FUNCTION_BLOCK FB_Idle IMPLEMENTS I_State
VAR_INPUT
	(* Pointer to the ATM Machine*)
	pATM_Machine	: POINTER TO FB_ATM_Machine;
END_VAR
VAR_OUTPUT
END_VAR
VAR
END_VAR

METHOD Cancel : BOOL
END_METHOD

METHOD Card_Ejected : BOOL
END_METHOD

METHOD Card_Inserted : BOOL
ADSLOGSTR(ADSLOG_MSGTYPE_LOG, 'Card has been inserted!', '');
pATM_Machine^.SetState(pATM_Machine^.ServingCustomerState);
END_METHOD

PROPERTY Description : E_StateDescription
GET
Description := E_StateDescription.Idle;
END_GET
END_PROPERTY

METHOD Failure : BOOL
END_METHOD

METHOD FB_Init : BOOL
VAR_INPUT
	(* if TRUE, the retain variables are initialized (warm start / cold start)*)
	bInitRetains	: BOOL;
	(* if TRUE, the instance afterwards gets moved into the copy code (online change)*)
	bInCopyCode	: BOOL;
	(* Pointer to the ATM Machine*)
	pATM_Machine	: POINTER TO FB_ATM_Machine;
END_VAR
THIS^.pATM_Machine := pATM_Machine;
END_METHOD

METHOD Op : BOOL
END_METHOD

METHOD Service : BOOL
ADSLOGSTR(ADSLOG_MSGTYPE_LOG, 'Entering Service Mode...', '');
pATM_Machine^.SetState(pATM_Machine^.MaintenanceState);
END_METHOD

METHOD SystemTest_OK : BOOL
END_METHOD

METHOD Turn_Off : BOOL
ADSLOGSTR(ADSLOG_MSGTYPE_LOG, 'Turning off machine...', '');
pATM_Machine^.SetState(pATM_Machine^.OffState);
END_METHOD

METHOD Turn_On : BOOL
END_METHOD

END_FUNCTION_BLOCK

(* stored: Version 1.1.0.1, ProductVersion 3.1.4024.12
   POU FB_Idle: Id {08375453-5d76-0934-1a95-46e42d833973}, SpecialFunc None
   Method Cancel: Id {65abf8fa-bea9-0656-26b8-1130a620e2a5}
   Method Card_Ejected: Id {529bb744-2dd3-091b-0da9-4215e7aa3d79}
   Method Card_Inserted: Id {4a45be97-fabb-0bf6-3e82-4d00f394dbe8}
   Property Description: Id {32d6cbbd-8d4f-077c-1475-851fe7226d1c}
   Get Get: Id {6ab89e4c-9a5b-0791-3189-ae0d014fa703}
   Method Failure: Id {1a918f8a-e3c3-04cc-3136-10375b9740ac}
   Method FB_Init: Id {c511d069-a148-0ad4-3acd-b9033977d1e7}
   Method Op: Id {d58a9927-21a9-057d-2612-bf7827879517}
   Method Service: Id {528a5b81-39cb-0ad8-390a-c4aba054ca09}
   Method SystemTest_OK: Id {4d033fde-e0c2-0cdc-2375-e8648799e634}
   Method Turn_Off: Id {67b1520e-2467-05df-32c1-7bd367dd3066}
   Method Turn_On: Id {7891db3f-3e8c-02e0-0648-e26dcab5460c} *)
